// Mitsubishi GX Works2 project: SEQUENCE_TIMER   PLC: Q03UDV

PROGRAM MAIN
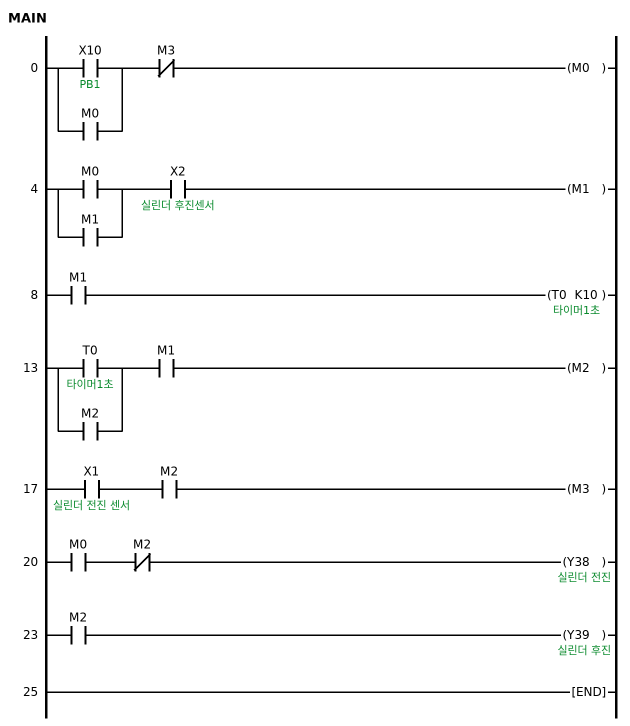
0     LD      X10  ; PB1
      OR      M0
      ANI     M3
      OUT     M0
4     LD      M0
      OR      M1
      AND     X2  ; 실린더 후진센서
      OUT     M1
8     LD      M1
      OUT     T0 K10  ; 타이머1초
13    LD      T0  ; 타이머1초
      OR      M2
      AND     M1
      OUT     M2
17    LD      X1  ; 실린더 전진 센서
      AND     M2
      OUT     M3
20    LD      M0
      ANI     M2
      OUT     Y38  ; 실린더 전진
23    LD      M2
      OUT     Y39  ; 실린더 후진
25    END
END_PROGRAM
